INTERFACE I_Motor

METHOD DrySpin : BOOL
VAR_INPUT
	nMotorSpeed : INT;
END_VAR
END_METHOD

METHOD ForwardSpin : BOOL
VAR_INPUT
	nMotorSpeed : INT;
END_VAR
END_METHOD

METHOD Stop : BOOL
VAR_INPUT
END_VAR
END_METHOD

END_INTERFACE

(* stored: Version 1.1.0.1, ProductVersion 3.1.4024.16
   Itf I_Motor: Id {926770be-804f-46bd-b05e-5e636180ea19}
   Method DrySpin: Id {2d17a97c-320f-442a-b73f-4d22dc8dd440}
   Method ForwardSpin: Id {42bbddb8-6174-49a2-9ced-f394ddff1965}
   Method Stop: Id {985aa12f-6584-4cba-b670-0479dc0cbaf6} *)
